# EPICS autosave request: NWPRTXPS/iocBoot/iocNWPRTXPS-IOC-01/NWPRTXPS_01_settings.req
# Motor settings
file "motor_settings.req" P=$(P), M=MTR$(CCP)01
file "motor_settings.req" P=$(P), M=MTR$(CCP)02
file "motor_settings.req" P=$(P), M=MTR$(CCP)03
file "motor_settings.req" P=$(P), M=MTR$(CCP)04
